// TIA Portal project "Urban Intersection Control System" (V17)

(* hardware
DEVICE "S7-1500/ET200MP station_1"  S7-1500 station
   slot 0: "Rail_0"  Rack  6ES7 590-1***0-0AA0
   slot 1: "PLC_UICS_01"  CPU 1512C-1 PN  6ES7 512-1CK00-0AB0  V2.9
      slot 3: "CPU display_1"  6ES7591-1AA00-0AA0
      slot 32768: "PROFINET interface_1"  X1
         slot 32769: "Port_1"  X1 P1
         slot 32770: "Port_2"  X1 P2
      slot 34817: "Virtual CP interface port_1"  Virtual CP interface port  Virtual CP interface port
*)

// ===== PLC "PLC_UICS_01"  CPU 1512C-1 PN =====

VAR_GLOBAL   // PLC tag table "UICS_Table"
   "PB_Ped_Main" AT %I10.2 : Bool;   // Push button for pedestrian crossing on Main Street
   "PB_Ped_Cross" AT %I10.3 : Bool;   // Push button for pedestrian crossing on Cross Street
   "EM_Main_Override" AT %I10.4 : Bool;   // Emergency override signal (e.g. ambulances) on Main Street
   "EM_Cross_Override" AT %I10.5 : Bool;   // Emergency override signal on Cross Street
   "SENSOR_Main_Vehicle" AT %I10.6 : Bool;   // Vehicle detection sensor on Main Street
   "SENSOR_Cross_Vehicle" AT %I10.7 : Bool;   // Vehicle detection sensor on Cross Street
   "TL_Main_Red" AT %Q4.0 : Bool;   // Red traffic light signal for Main Street
   "TL_Main_Yellow" AT %Q4.1 : Bool;   // Yellow traffic light signal for Main Street
   "TL_Main_Green" AT %Q4.2 : Bool;   // Green traffic light signal for Main Street
   "TL_Cross_Red" AT %Q4.3 : Bool;   // Red traffic light signal for Cross Street
   "TL_Cross_Yellow" AT %Q4.4 : Bool;   // Yellow traffic light signal for Cross Street
   "TL_Cross_Green" AT %Q4.5 : Bool;   // Green traffic light signal for Cross Street
   "PED_Main_Walk" AT %Q4.6 : Bool;   // Pedestrian walk signal for Main Street
   "PED_Main_Dontwalk" AT %Q4.7 : Bool;   // Pedestrian don’t-walk signal for Main Street
   "PED_Cross_Walk" AT %Q5.0 : Bool;   // Pedestrian walk signal for Cross Street
   "PED_Cross_DontWalk" AT %Q5.1 : Bool;   // Pedestrian don’t-walk signal for Cross Street
   "PED_Warning_Buzzer" AT %Q5.2 : Bool;   // Audible alert for pedestrian crossing
   "SYS_Stop" AT %I10.1 : Bool;   // Emergency stop function
   "SYS_Start" AT %I10.0 : Bool;   // Begins the system
END_VAR

DATA_BLOCK "Main_Control_System_DB"   // DB1
{ S7_Optimized_Access := 'TRUE' }
VERSION : 0.1
// stored: InstanceOfName Main_Control_System
"Main_Control_System"
BEGIN
END_DATA_BLOCK

// folder: System blocks/Program resources

DATA_BLOCK "Red_Timer_DB"   // DB2
{ S7_Optimized_Access := 'TRUE' }
AUTHOR : Simatic
FAMILY : IEC
NAME : IEC_TMR
VERSION : 1.0
// stored: InstanceOfName IEC_TIMER
"IEC_TIMER"
BEGIN
END_DATA_BLOCK

DATA_BLOCK "Green_Timer_DB"   // DB3
{ S7_Optimized_Access := 'TRUE' }
AUTHOR : Simatic
FAMILY : IEC
NAME : IEC_TMR
VERSION : 1.0
// stored: InstanceOfName IEC_TIMER
"IEC_TIMER"
BEGIN
END_DATA_BLOCK

DATA_BLOCK "Yellow_Timer_DB"   // DB4
{ S7_Optimized_Access := 'TRUE' }
AUTHOR : Simatic
FAMILY : IEC
NAME : IEC_TMR
VERSION : 1.0
// stored: InstanceOfName IEC_TIMER
"IEC_TIMER"
BEGIN
END_DATA_BLOCK

// folder: (top level)

FUNCTION_BLOCK "Main_Control_System"   // FB1, LAD
{ S7_Optimized_Access := 'TRUE' }
VERSION : 0.1
   VAR
      System_Running : Bool;   // System is actively running
      Emergency_Stop : Bool;   // Emergency stop activated flag
   END_VAR
BEGIN

REGION Network 1: Main Street Traffic
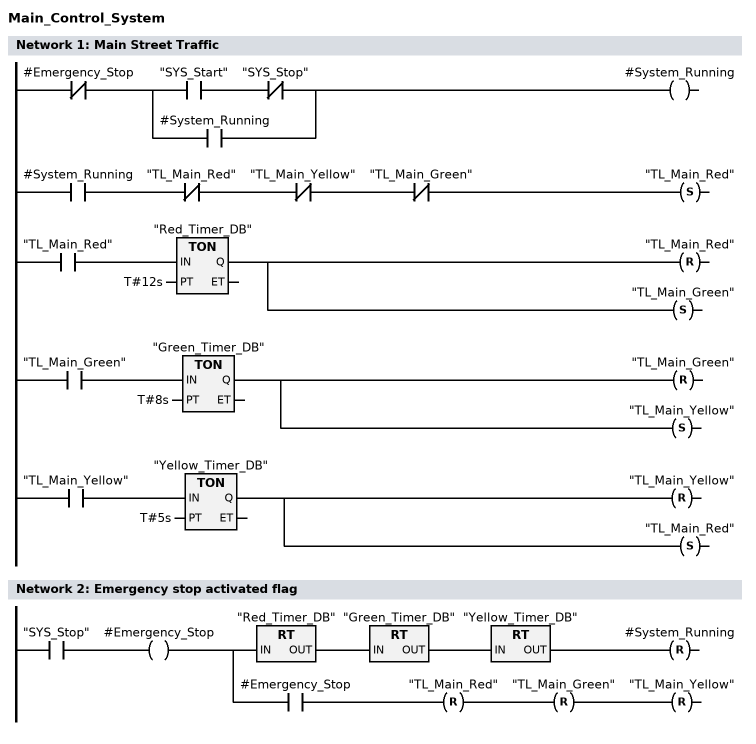
   #System_Running := NOT #Emergency_Stop AND (("SYS_Start" AND NOT "SYS_Stop") OR #System_Running);
   IF #System_Running AND NOT "TL_Main_Red" AND NOT "TL_Main_Yellow" AND NOT "TL_Main_Green" THEN
       "TL_Main_Red" := TRUE;
   END_IF;
   "Red_Timer_DB".TON(IN := "TL_Main_Red", PT := T#12s);
   IF "Red_Timer_DB".Q THEN
       "TL_Main_Red" := FALSE;
       "TL_Main_Green" := TRUE;
   END_IF;
   "Green_Timer_DB".TON(IN := "TL_Main_Green", PT := T#8s);
   IF "Green_Timer_DB".Q THEN
       "TL_Main_Green" := FALSE;
       "TL_Main_Yellow" := TRUE;
   END_IF;
   "Yellow_Timer_DB".TON(IN := "TL_Main_Yellow", PT := T#5s);
   IF "Yellow_Timer_DB".Q THEN
       "TL_Main_Yellow" := FALSE;
       "TL_Main_Red" := TRUE;
   END_IF;
END_REGION

REGION Network 2: Emergency stop activated flag
   RUNG wire#powerrail
      Contact( "SYS_Stop" )
      Coil( #Emergency_Stop )
      wire#w1
      RT_Coil( "Red_Timer_DB" )
      RT_Coil( "Green_Timer_DB" )
      RT_Coil( "Yellow_Timer_DB" )
      R_Coil( #System_Running )
   END_RUNG
   RUNG wire#w1
      Contact( #Emergency_Stop )
      R_Coil( "TL_Main_Red" )
      R_Coil( "TL_Main_Green" )
      R_Coil( "TL_Main_Yellow" )
   END_RUNG
   // the same network as SCL:
   #Emergency_Stop := "SYS_Stop";
   IF "SYS_Stop" THEN
       RESET_TIMER("Red_Timer_DB");
       RESET_TIMER("Green_Timer_DB");
       RESET_TIMER("Yellow_Timer_DB");
       #System_Running := FALSE;
   END_IF;
   IF "SYS_Stop" AND #Emergency_Stop THEN
       "TL_Main_Red" := FALSE;
       "TL_Main_Green" := FALSE;
       "TL_Main_Yellow" := FALSE;
   END_IF;
END_REGION
END_FUNCTION_BLOCK

ORGANIZATION_BLOCK "Main"   // OB1, LAD, ProgramCycle
TITLE = "Main Program Sweep (Cycle)"
{ S7_Optimized_Access := 'TRUE' }
VERSION : 0.1
   VAR_INPUT
      Initial_Call : Bool;   // Initial call of this OB
      Remanence : Bool;   // =True, if remanent data are available
   END_VAR
BEGIN

REGION Network 1: Main
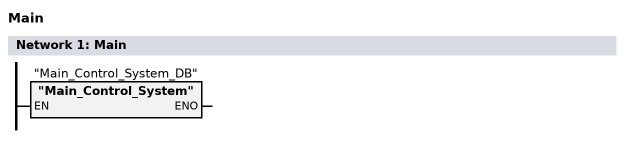
   RUNG wire#powerrail
      "Main_Control_System_DB"()
   END_RUNG
   // the same network as SCL:
   "Main_Control_System_DB"();   // "Main_Control_System"
END_REGION
END_ORGANIZATION_BLOCK